Universal Robots PolyScope program: KZXD.urp

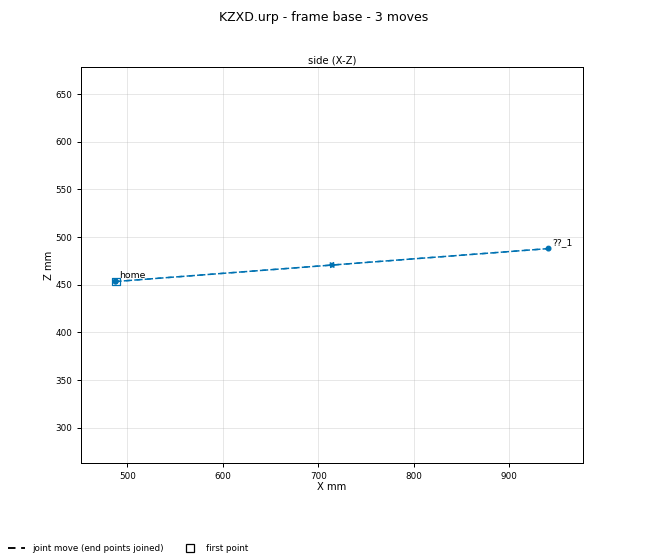
[picture p0: tool path of KZXD.urp in frame base, 3 of 3 moves have a stored position in this frame; points joined in program order, loops and branches not executed]
Program KZXD (installation=default directory=/programs/usbdisk createdIn=3.11.0.82155 lastSavedIn=3.11.0.82155 robotSerialNumber=2019301986)
Calibrated DH parameters: a=[-0.000016, -0.608674, -0.475969, 0.000036, 0.000098, 0]; d=[0.128083, 6.301652, -136.10008, 129.961951, 0.115705, 0.092166]; alpha=[1.570916, -0.010815, -0.002431, 1.570538, -1.573046, 0]; deltaTheta=[-0.000061, -0.111545, 0.697038, -0.585376, -0.000066, 0.000029]
Robot Program (runOnlyOnce=true)
  Set DigitalOutput pin=digital_out[1]; digitalValue=0
  MoveJ speed 60 deg/s, acceleration 80 deg/s^2 (useActiveTCP=true)
    Waypoint home: TCP in base x=487.593 y=103.241 z=453.444 mm, rx=-1.7356 ry=0.7158 rz=-1.7079 rad; joints [-190.105, -92.975, 137.713, -225.032, -77.949, -42.611] deg
    Waypoint 路点_1: TCP in base x=941.574 y=103.268 z=487.983 mm, rx=-2.847 ry=1.2456 rz=0.0439 rad; joints [-184.347, -65.232, 75.668, -99.702, -87.918, -46.593] deg
    Wait Sleep waitTime=20
  Loop Counting (count=3) loopVariable(name=循环_1)
    Set DigitalOutput pin=digital_out[0]; digitalValue=1
    Pallet pattern(dimensionality=Line firstAxisCount=3 secondAxisCount=5 thirdAxisCount=5 motionType=MoveL speed=0.25 acceleration=1.2 useActiveTCP=true, counterVariable(name=cnt_1, initializeExpression=0), patternPoseVariable(name=位姿_1), feature=Base, children(Waypoint(type=Fixed name=起始位置_1, position(joints=-2.8679118792163294, -0.6052992979632776, 0.9743008613586426, -1.9209817091571253, -1.5607226530658167, -0.4844926039325159 pose=1.0601035283906166, 0.4754525613910999, 0.17781263736057795, -2.887209323466087, 1.233162646415982, 0.0450490158549316), poseInFeatureCoordinates=[1.060104, 0.475453, 0.177813, -2.887209, 1.233163, 0.045049], outputFlangePose=[1.060104, 0.475453, 0.177813, -2.887209, 1.233163, 0.045049]), Waypoint(type=Fixed name=终止位置_1, position(joints=-3.8029587904559534, -0.46518165269960576, 0.7185640335083008, -1.7983410994159144, -1.5868366400348108, -1.420300308858053 pose=1.0600769881298873, -0.6122792094126899, 0.16625052380852423, -2.887264695427694, 1.233098884871615, 0.04501916540262987), poseInFeatureCoordinates=[1.060077, -0.612279, 0.166251, -2.887265, 1.233099, 0.045019], outputFlangePose=[1.060077, -0.612279, 0.166251, -2.887265, 1.233099, 0.045019]))); actionSequence(name=托盘序列 motionType=MoveL speed=0.25 acceleration=1.2 useActiveTCP=true, anchorWaypoint(type=Fixed name=模式点_1, position(joints=-2.8679238001452845, -0.605323616658346, 0.9743247032165527, -1.9210298697101038, -1.5607107321368616, -0.48454028764833623 pose=1.060105201596643, 0.47543999361233347, 0.17783066240786258, -2.8871946990368937, 1.2330951645032995, 0.04500073620475842), poseInFeatureCoordinates=[1.060105, 0.47544, 0.177831, -2.887195, 1.233095, 0.045001], outputFlangePose=[1.060105, 0.47544, 0.177831, -2.887195, 1.233095, 0.045001]), feature=Base, children(Waypoint(type=Fixed name=方式, position(joints=-2.8679238001452845, -0.6437371412860315, 0.9383525848388672, -1.8468650023089808, -1.5606029669391077, -0.48402530351747686 pose=1.0601503747853316, 0.475394959391514, 0.237069360703778, -2.887040274070396, 1.233198936194579, 0.04470252865491039), poseInFeatureCoordinates=[1.06015, 0.475395, 0.237069, -2.88704, 1.233199, 0.044703], outputFlangePose=[1.06015, 0.475395, 0.237069, -2.88704, 1.233199, 0.044703]), Waypoint=模式点_1, Set(type=NoAction), SuppressedNode(suppressedNode(type=Sleep, waitTime=180)), Waypoint(type=Fixed name=退出, position(joints=-2.8679118792163294, -0.6437371412860315, 0.9383525848388672, -1.8468287626849573, -1.5605428854571741, -0.48407298723329717 pose=1.0601398845155643, 0.4754120142343888, 0.23706534030971022, -2.887053064588625, 1.2331035295624941, 0.044805787690121585), poseInFeatureCoordinates=[1.06014, 0.475412, 0.237065, -2.887053, 1.233104, 0.044806], outputFlangePose=[1.06014, 0.475412, 0.237065, -2.887053, 1.233104, 0.044806])))
      Pattern -> pattern
      AnchoredSequence -> 托盘序列
  Set DigitalOutput pin=digital_out[0]; digitalValue=0
  SuppressedNode
    Wait Sleep waitTime=300
  MoveJ speed 60 deg/s, acceleration 80 deg/s^2 (useActiveTCP=true)
    Waypoint 路点_2: TCP in base x=487.599 y=103.2 z=453.463 mm, rx=-1.7356 ry=0.7159 rz=-1.7079 rad; joints [-190.111, -92.977, 137.712, -225.03, -77.947, -42.611] deg
  Set DigitalOutput pin=digital_out[1]; digitalValue=1
